// TIA Portal V18 export
DATA_BLOCK "Aux_Motor_Control_DB"   // DB12
// stored: AutoNumber false, InstanceOfName Aux_Motor_Control, InstanceOfType FB
"Aux_Motor_Control"
   // VAR
   //    AuxPumpStartTOF { S7_SetPoint := 'True'} : TOF_TIME;
   //    AuxPumpFailTON { S7_SetPoint := 'True'} : TON_TIME;
   //    CoolingFanFailTON { S7_SetPoint := 'True'} : TON_TIME;
   //    CoolingFanStartTON { S7_SetPoint := 'True'} : TOF_TIME;
   // END_VAR
BEGIN
END_DATA_BLOCK
